Universal Robots PolyScope program: motor_plate_positioning_example.urp

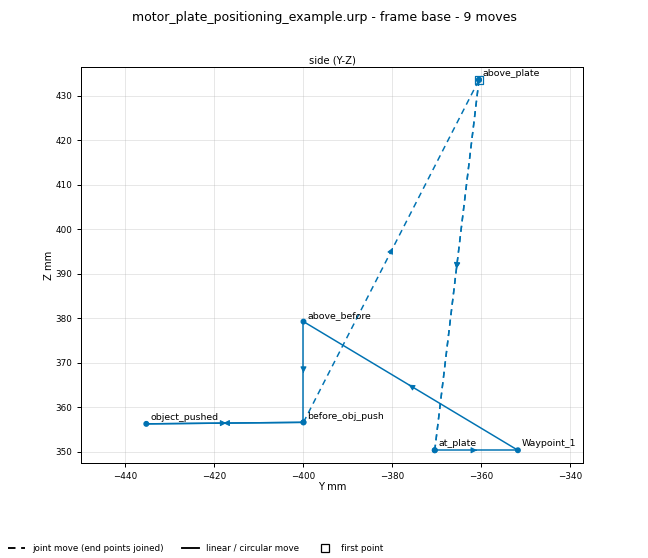
[picture p0: tool path of motor_plate_positioning_example.urp in frame base, 9 of 9 moves have a stored position in this frame; points joined in program order, loops and branches not executed]
Program motor_plate_positioning_example (installation=default directory=/programs/wrs2020 createdIn=5.6.0.90886 lastSavedIn=5.9.1.1031110 robotSerialNumber=20205500180)
Calibrated DH parameters: a=[0, -0.425, -0.3922, 0, 0, 0]; d=[0.1625, 0, 0, 0.1333, 0.0997, 0.0996]; alpha=[1.570796, 0, 0, 1.570796, -1.570796, 0]; deltaTheta=[0, 0, 0, 0, 0, 0]
Robot Program (runOnlyOnce=true)
  URCap Gripper (Robotiq_Grippers, Robotiq Inc.) dataModel(position=58.8235294117647, force=0.0, speed=0.0, positionInDouble=58.8235294117647, forceInDouble=0.0, speedInDouble=0.0, slaveIds=[9], blocking=true)
  MoveJ speed 60 deg/s, acceleration 80 deg/s^2 (useActiveTCP=false) tcp=TCP; feature=Base
    Waypoint above_plate: TCP in base x=113.193 y=-360.458 z=433.533 mm, rx=0.0037 ry=3.0617 rz=-0.699 rad; joints [86.404, -112.982, 123.786, -126.397, -88.216, -3.05] deg
    Waypoint at_plate: TCP in base x=113.193 y=-370.401 z=350.29 mm, rx=0.0037 ry=3.0617 rz=-0.699 rad; joints [86.494, -106.791, 132.85, -141.656, -88.265, -2.917] deg
  URCap Gripper (Robotiq_Grippers, Robotiq Inc.) dataModel(position=100.0, force=0.0, speed=0.0, positionInDouble=100.0, forceInDouble=0.0, speedInDouble=0.0, slaveIds=[9], blocking=true)
  Popup Message (haltProgram=false message=start? inputType=Text)
  MoveL speed 250 mm/s, acceleration 1200 mm/s^2 (useActiveTCP=false) tcp=TCP; feature=Base
    Waypoint Waypoint_1: TCP in base x=113.193 y=-351.716 z=350.29 mm, rx=0.0037 ry=3.0617 rz=-0.699 rad; joints [86.282, -110.025, 134.858, -140.425, -88.171, -3.116] deg
  URCap Gripper (Robotiq_Grippers, Robotiq Inc.) dataModel(position=72.54901960784314, force=0.0, speed=0.0, positionInDouble=72.54901960784314, forceInDouble=0.0, speedInDouble=0.0, slaveIds=[9], blocking=true)
  MoveL speed 250 mm/s, acceleration 1200 mm/s^2 (useActiveTCP=false) tcp=TCP; feature=Base
    Waypoint above_before: TCP in base x=113.226 y=-399.906 z=379.207 mm, rx=0.004 ry=3.141 rz=0.0154 rad; joints [87.175, -101.487, 116.102, -103.97, -89.821, -2.686] deg
    Waypoint before_obj_push: TCP in base x=113.226 y=-399.906 z=356.565 mm, rx=0.004 ry=3.141 rz=0.0154 rad; joints [87.172, -100.511, 118.783, -107.626, -89.818, -2.678] deg
  URCap Gripper (Robotiq_Grippers, Robotiq Inc.) dataModel(position=100.0, force=0.0, speed=0.0, positionInDouble=100.0, forceInDouble=0.0, speedInDouble=0.0, slaveIds=[9], blocking=true)
  MoveL speed 250 mm/s, acceleration 1200 mm/s^2 (useActiveTCP=false) tcp=TCP; feature=Base
    Waypoint object_pushed: motionParameters(jointSpeed=1.047198 jointAcceleration=1.396263 cartesianSpeed=0.008 cartesianAcceleration=1.2); TCP in base x=113.139 y=-435.23 z=356.222 mm, rx=0.004 ry=3.141 rz=0.0154 rad; joints [87.384, -95.381, 114.516, -108.489, -89.814, -2.455] deg
    Waypoint before_obj_push: TCP in base x=113.226 y=-399.906 z=356.565 mm, rx=0.004 ry=3.141 rz=0.0154 rad; joints [87.172, -100.511, 118.783, -107.626, -89.818, -2.678] deg
  URCap Gripper (Robotiq_Grippers, Robotiq Inc.) dataModel(position=72.54901960784314, force=0.0, speed=0.0, positionInDouble=72.54901960784314, forceInDouble=0.0, speedInDouble=0.0, slaveIds=[9], blocking=true)
  MoveJ speed 60 deg/s, acceleration 80 deg/s^2 (useActiveTCP=false) tcp=TCP; feature=Base
    Waypoint above_plate: TCP in base x=113.193 y=-360.458 z=433.533 mm, rx=0.0037 ry=3.0617 rz=-0.699 rad; joints [86.404, -112.982, 123.786, -126.397, -88.216, -3.05] deg
    Waypoint at_plate: TCP in base x=113.193 y=-370.401 z=350.29 mm, rx=0.0037 ry=3.0617 rz=-0.699 rad; joints [86.494, -106.791, 132.85, -141.656, -88.265, -2.917] deg
  URCap Gripper (Robotiq_Grippers, Robotiq Inc.) dataModel(position=100.0, force=0.0, speed=0.0, positionInDouble=100.0, forceInDouble=0.0, speedInDouble=0.0, slaveIds=[9], blocking=true)
